// SIMATIC S7-200 project (STEP 7-Micro/WIN), CPU 222 REL 02.01

ORGANIZATION_BLOCK MAIN:OB1
TITLE=PROGRAM COMMENTS
BEGIN
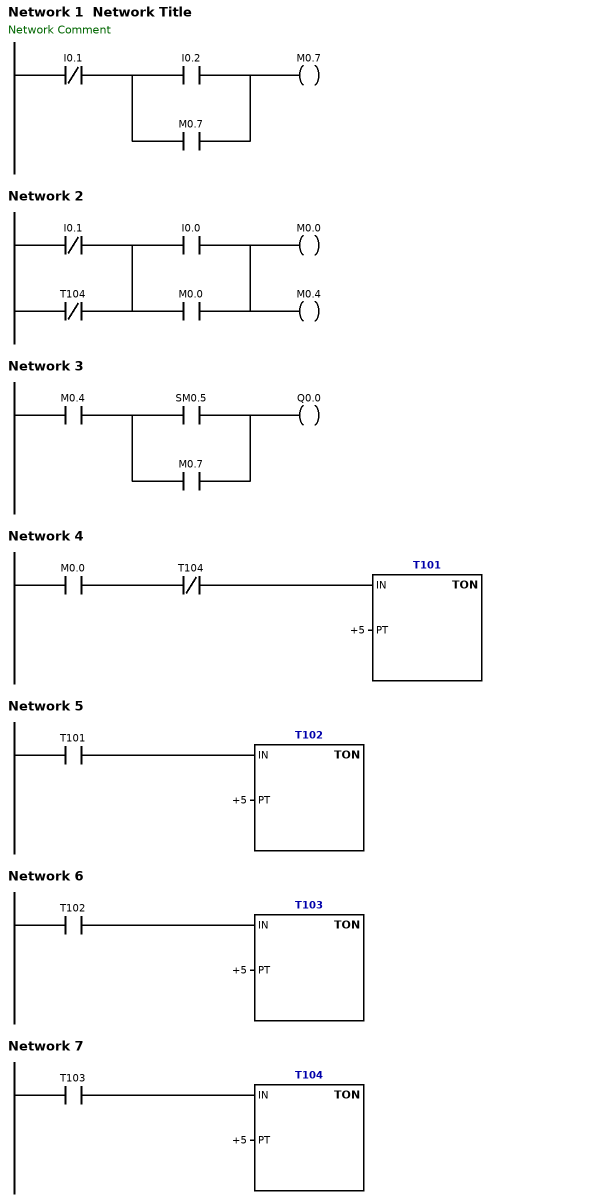
Network 1 // Network Title
// Network Comment
LDN    I0.1
LD     I0.2
O      M0.7
ALD
=      M0.7
Network 2
LDN    I0.1
ON     T104
LD     I0.0
O      M0.0
ALD
=      M0.0
=      M0.4
Network 3
LD     M0.4
LD     SM0.5
O      M0.7
ALD
=      Q0.0
Network 4
LD     M0.0
AN     T104
TON    T101, +5
Network 5
LD     T101
TON    T102, +5
Network 6
LD     T102
TON    T103, +5
Network 7
LD     T103
TON    T104, +5
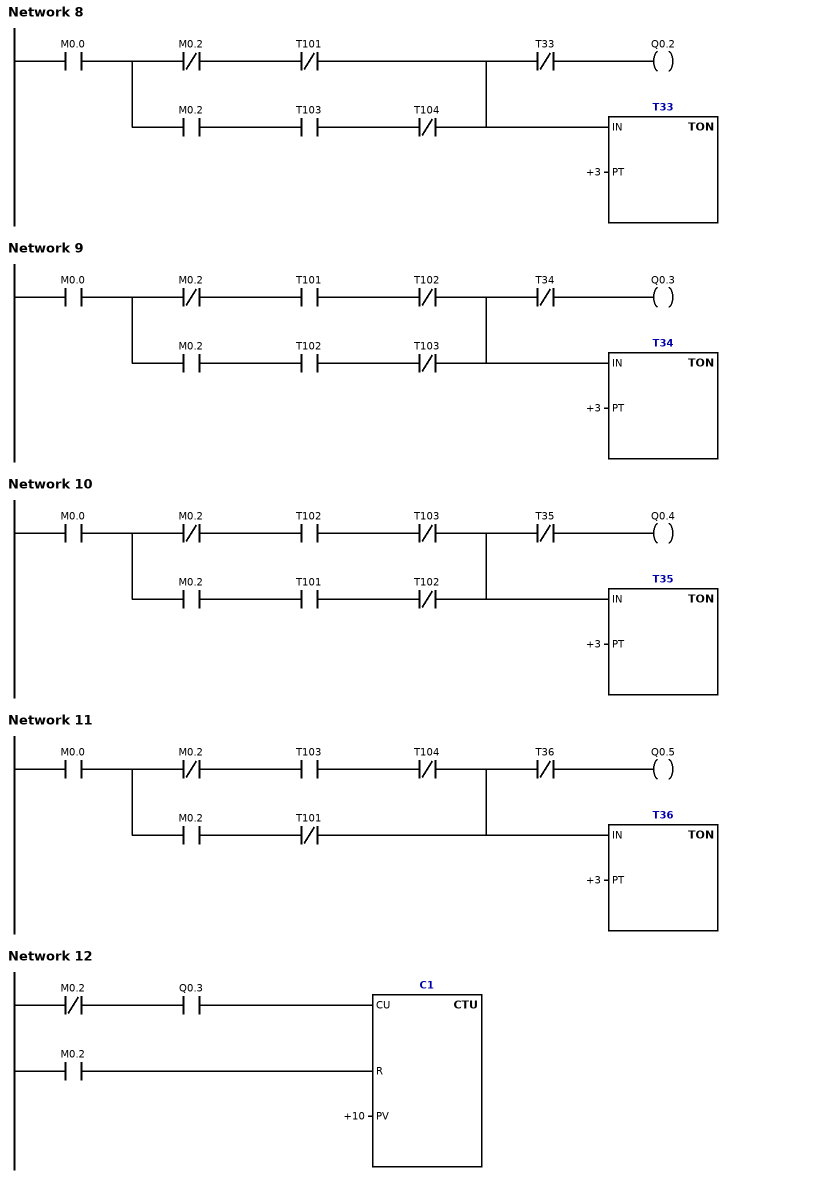
Network 8
LD     M0.0
LDN    M0.2
AN     T101
LD     M0.2
A      T103
AN     T104
OLD
ALD
LPS
AN     T33
=      Q0.2
LPP
TON    T33, +3
Network 9
LD     M0.0
LDN    M0.2
A      T101
AN     T102
LD     M0.2
A      T102
AN     T103
OLD
ALD
LPS
AN     T34
=      Q0.3
LPP
TON    T34, +3
Network 10
LD     M0.0
LDN    M0.2
A      T102
AN     T103
LD     M0.2
A      T101
AN     T102
OLD
ALD
LPS
AN     T35
=      Q0.4
LPP
TON    T35, +3
Network 11
LD     M0.0
LDN    M0.2
A      T103
AN     T104
LD     M0.2
AN     T101
OLD
ALD
LPS
AN     T36
=      Q0.5
LPP
TON    T36, +3
Network 12
LDN    M0.2
A      Q0.3
LD     M0.2
CTU    C1, +10
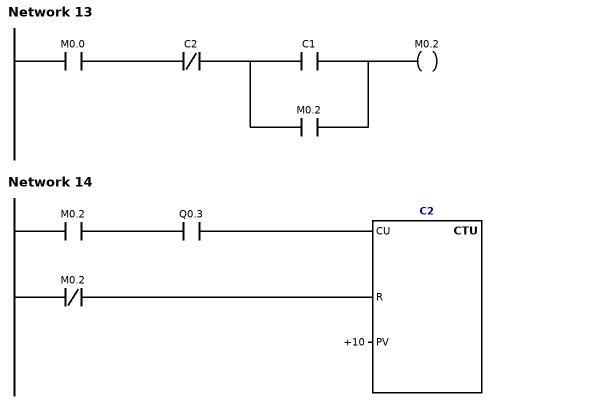
Network 13
LD     M0.0
AN     C2
LD     C1
O      M0.2
ALD
=      M0.2
Network 14
LD     M0.2
A      Q0.3
LDN    M0.2
CTU    C2, +10
END_ORGANIZATION_BLOCK
